// TIA Portal V19 export
ORGANIZATION_BLOCK "Main"   // OB1, LAD, ProgramCycle
TITLE = "Main Program Sweep (Cycle)"
{ S7_Optimized_Access := 'TRUE' }
// stored: SetENOAutomatically false
   VAR_INPUT
      Initial_Call : Bool;   // Initial call of this OB
      Remanence : Bool;   // =True, if remanent data are available
   END_VAR
BEGIN

REGION Network 1
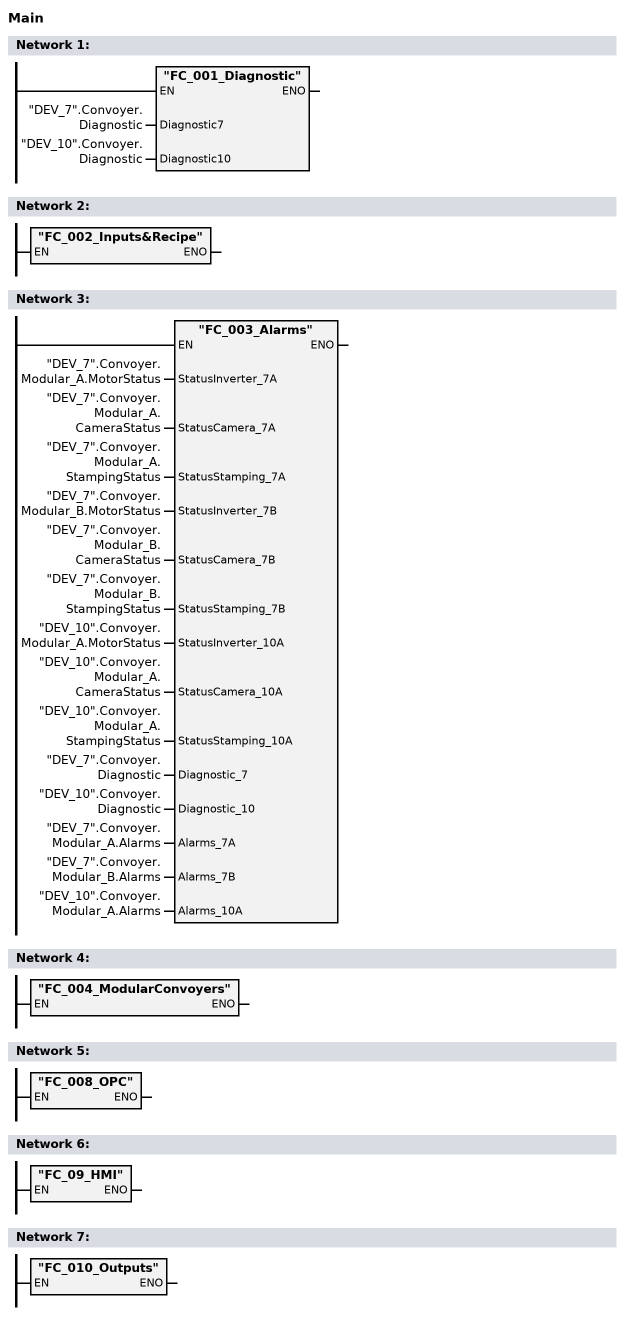
   RUNG wire#powerrail
      "FC_001_Diagnostic"(Diagnostic7 := "DEV_7".Convoyer.Diagnostic, Diagnostic10 := "DEV_10".Convoyer.Diagnostic)
   END_RUNG
   // the same network as SCL:
   "FC_001_Diagnostic"(Diagnostic7 := "DEV_7".Convoyer.Diagnostic, Diagnostic10 := "DEV_10".Convoyer.Diagnostic);
END_REGION

REGION Network 2
   RUNG wire#powerrail
      "FC_002_Inputs&Recipe"()
   END_RUNG
   // the same network as SCL:
   "FC_002_Inputs&Recipe"();
END_REGION

REGION Network 3
   RUNG wire#powerrail
      "FC_003_Alarms"(StatusInverter_7A := "DEV_7".Convoyer.Modular_A.MotorStatus, StatusCamera_7A := "DEV_7".Convoyer.Modular_A.CameraStatus, StatusStamping_7A := "DEV_7".Convoyer.Modular_A.StampingStatus, StatusInverter_7B := "DEV_7".Convoyer.Modular_B.MotorStatus, StatusCamera_7B := "DEV_7".Convoyer.Modular_B.CameraStatus, StatusStamping_7B := "DEV_7".Convoyer.Modular_B.StampingStatus, StatusInverter_10A := "DEV_10".Convoyer.Modular_A.MotorStatus, StatusCamera_10A := "DEV_10".Convoyer.Modular_A.CameraStatus, StatusStamping_10A := "DEV_10".Convoyer.Modular_A.StampingStatus, Diagnostic_7 := "DEV_7".Convoyer.Diagnostic, Diagnostic_10 := "DEV_10".Convoyer.Diagnostic, Alarms_7A := "DEV_7".Convoyer.Modular_A.Alarms, Alarms_7B := "DEV_7".Convoyer.Modular_B.Alarms, Alarms_10A := "DEV_10".Convoyer.Modular_A.Alarms)
   END_RUNG
   // the same network as SCL:
   "FC_003_Alarms"(StatusInverter_7A := "DEV_7".Convoyer.Modular_A.MotorStatus,
                   StatusCamera_7A := "DEV_7".Convoyer.Modular_A.CameraStatus,
                   StatusStamping_7A := "DEV_7".Convoyer.Modular_A.StampingStatus,
                   StatusInverter_7B := "DEV_7".Convoyer.Modular_B.MotorStatus,
                   StatusCamera_7B := "DEV_7".Convoyer.Modular_B.CameraStatus,
                   StatusStamping_7B := "DEV_7".Convoyer.Modular_B.StampingStatus,
                   StatusInverter_10A := "DEV_10".Convoyer.Modular_A.MotorStatus,
                   StatusCamera_10A := "DEV_10".Convoyer.Modular_A.CameraStatus,
                   StatusStamping_10A := "DEV_10".Convoyer.Modular_A.StampingStatus,
                   Diagnostic_7 := "DEV_7".Convoyer.Diagnostic,
                   Diagnostic_10 := "DEV_10".Convoyer.Diagnostic,
                   Alarms_7A := "DEV_7".Convoyer.Modular_A.Alarms,
                   Alarms_7B := "DEV_7".Convoyer.Modular_B.Alarms,
                   Alarms_10A := "DEV_10".Convoyer.Modular_A.Alarms);
END_REGION

REGION Network 4
   RUNG wire#powerrail
      "FC_004_ModularConvoyers"()
   END_RUNG
   // the same network as SCL:
   "FC_004_ModularConvoyers"();
END_REGION

REGION Network 5
   RUNG wire#powerrail
      "FC_008_OPC"()
   END_RUNG
   // the same network as SCL:
   "FC_008_OPC"();
END_REGION

REGION Network 6
   RUNG wire#powerrail
      "FC_09_HMI"()
   END_RUNG
   // the same network as SCL:
   "FC_09_HMI"();
END_REGION

REGION Network 7
   RUNG wire#powerrail
      "FC_010_Outputs"()
   END_RUNG
   // the same network as SCL:
   "FC_010_Outputs"();
END_REGION
END_ORGANIZATION_BLOCK
